(* PLC project CoDeSys External Library Template, WAGO e!COCKPIT e!COCKPIT, author 3S - Smart Software Solutions GmbH *)
(* stored: creationDateTime 2019-10-29T12:22:40.7814712, version 3.5.5.30, modificationDateTime 2019-10-24T14:40:07.960949, organization 3S - Smart Software Solutions GmbH *)
(* Library project template with all possible element types, docu and a sample project structure *)

FUNCTION fnCRC16Obliczanie : WORD
  VAR_INPUT
    sKomunikat : alSTRINGKomunikat;
  END_VAR
  VAR
    intPetla : INT;
    wCRC16_modbus : WORD;
    arTransmitterBuffer : ARRAY[1..512] OF BYTE;
  END_VAR

            FOR intPetla := 1 TO LEN(sKomunikat) BY 1 DO
	arTransmitterBuffer[intPetla] := string_to_ASCIIByte(MID(sKomunikat , 1 , intPetla));
END_FOR

fnCRC16Obliczanie := MEM.CRC16_modbus(ADR(arTransmitterBuffer[1]) , INT_TO_UINT(LEN(sKomunikat)));
          
END_FUNCTION
